Yaskawa INFORM job: RECUA_PINOS.JBI

/JOB
//NAME RECUA_PINOS
///FOLDERNAME GRAMPOS
//POS
///NPOS 0,0,0,0,0,0
//INST
///DATE 2022/06/09 09:24
///ATTR SC,RW
NOP
DOUT OT#(539) OFF
DOUT OT#(540) ON
WAIT IN#(545)=ON
WAIT IN#(547)=ON
END
